SYSTEM ResourceDeploymentTest
  (* Version 1.0, 2024-08-21, mario *)
  APPLICATION ResourceDeploymentTestApp
  END_APPLICATION
  DEVICE FORTE_PC : FORTE_PC(MGR_ID := "localhost:61499" (* Device manager socket ID *))
    {SET_ATTRIBUTE(Profile, HOLOBLOC)}
    RESOURCE TestNumberOfParams : EMB_RES
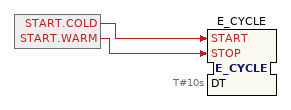
      FBS
        E_CYCLE : E_CYCLE(DT := T#10s);
      END_FBS
      EVENT_CONNECTIONS
        START.COLD TO E_CYCLE.START;
        START.WARM TO E_CYCLE.STOP;
      END_CONNECTIONS
    END_RESOURCE
    RESOURCE TestParamsIdentity : EMB_RES
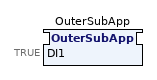
      SUBAPPS
        OuterSubApp : OuterSubApp(DI1 := TRUE);
      END_SUBAPPS
    END_RESOURCE
  END_DEVICE
END_SYSTEM
